# EPICS StreamDevice protocol: protocols/bwg.proto
Terminator = LF;
ExtraInput = Ignore;

setNCO {
	out "w\${1}_nco %d";
	in;
}

setLEN {
	out "w\${1}_len %d";
	in;
}

setENABLE {
	out "w\${1}_cr %d";
	in;
}

getReps {
	out "w\${1}_sta";
	in "%d,%*d";
}

getNcoClk {
	out "w\${1}_sta";
	in "%*d,%d";
}
